// TIA Portal V17 export
// export: Created 2023-02-13T11:16:08.4914499Z, ExportSetting WithDefaults, DisplayName Totally Integrated Automation Portal, DisplayVersion V17, DisplayName TIA Portal Openness, DisplayVersion V17, DisplayName TIA Portal Teamcenter Gateway, DisplayVersion V17, DisplayName TIA Portal Version Control Interface, DisplayVersion V17, DisplayName SINAMICS Startdrive Advanced, DisplayVersion V17, DisplayName SINAMICS Startdrive G130, G150, S120, S150, SINAMICS MV, S210, DisplayVersion V17, DisplayName SINAMICS Startdrive G110M, G120, G120C, G120D, G120P, G115D, DisplayVersion V17, DisplayName STEP 7 Professional, DisplayVersion V17, DisplayName STEP 7 Safety, DisplayVersion V17, DisplayName WinCC Professional, DisplayVersion V17
FUNCTION_BLOCK "Alarm Flow Collector"   // FB211, LAD
{ S7_Optimized_Access := 'TRUE' }
VERSION : 0.1
// stored: AutoNumber false, IsIECCheckEnabled false, IsRetainMemResEnabled false, MemoryReserve 100, SetENOAutomatically false, UDAEnableTagReadback false
   VAR_INPUT
      Reset : Bool;
   END_VAR
   VAR
      alwaysON : Bool;
   END_VAR
   VAR RETAIN
      Param : Struct
         min_Flow : Struct
            ChiliAwetan1 : Real := 5.0;
            ChiliAwetan2 : Real := 5.0;
            ChiliAwetan3 : Real := 5.0;
            Tomato : Real := 5.0;
            ChiliFresh1 : Real := 5.0;
            ChiliFresh2 : Real := 5.0;
            ChiliFresh3 : Real := 5.0;
            Garlic : Real := 5.0;
            HW : Real := 5.0;
            Vinegar : Real := 5.0;
            Sugar : Real := 5.0;
            Salt : Real := 5.0;
            ProWater : Real := 5.0;
            Homomixer : Real := 5.0;
         END_STRUCT;
         timerMon : Struct
            ChiliAwetan1 : TON_TIME;
            ChiliAwetan2 : TON_TIME;
            ChiliAwetan3 : TON_TIME;
            Tomato : TON_TIME;
            ChiliFresh1 : TON_TIME;
            ChiliFresh2 : TON_TIME;
            ChiliFresh3 : TON_TIME;
            Garlic : TON_TIME;
            HW : TON_TIME;
            Vinegar : TON_TIME;
            Sugar : TON_TIME;
            Salt : TON_TIME;
            ProWater : TON_TIME;
            Homomixer : TON_TIME;
         END_STRUCT;
      END_STRUCT;
   END_VAR
   VAR
      AlarmFlow_Blend : Word;
   END_VAR
   // Param.timerMon.ChiliAwetan1.PT := T#20s;
   // Param.timerMon.ChiliAwetan2.PT := T#20s;
   // Param.timerMon.ChiliAwetan3.PT := T#20s;
   // Param.timerMon.Tomato.PT := T#20s;
   // Param.timerMon.ChiliFresh1.PT := T#20s;
   // Param.timerMon.ChiliFresh2.PT := T#20s;
   // Param.timerMon.ChiliFresh3.PT := T#20s;
   // Param.timerMon.Garlic.PT := T#20s;
   // Param.timerMon.HW.PT := T#20s;
   // Param.timerMon.Vinegar.PT := T#20s;
   // Param.timerMon.Sugar.PT := T#20s;
   // Param.timerMon.Salt.PT := T#20s;
   // Param.timerMon.ProWater.PT := T#20s;
   // Param.timerMon.Homomixer.PT := T#20s;
BEGIN

REGION Network 1: always ON
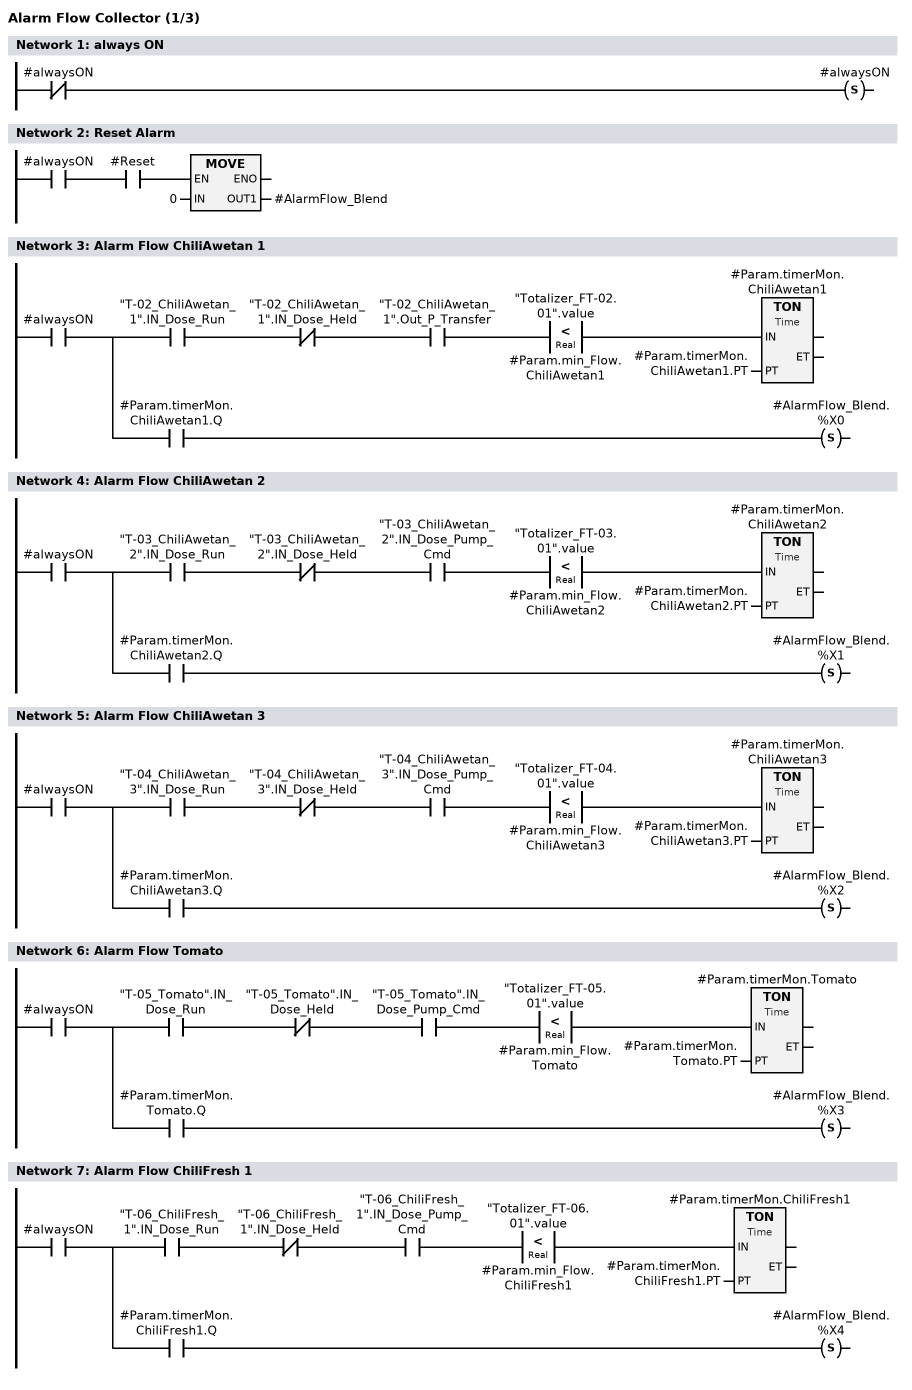
   RUNG wire#powerrail
      I_Contact( #alwaysON )
      S_Coil( #alwaysON )
   END_RUNG
   // the same network as SCL:
   IF NOT #alwaysON THEN #alwaysON := TRUE; END_IF;
END_REGION

REGION Network 2: Reset Alarm
   RUNG wire#powerrail
      Contact( #alwaysON )
      Contact( #Reset )
      Move(in := 0, out1 => #AlarmFlow_Blend)
   END_RUNG
   // the same network as SCL:
   IF #alwaysON AND #Reset THEN #AlarmFlow_Blend := 0; END_IF;
END_REGION

REGION Network 3: Alarm Flow ChiliAwetan 1
   RUNG wire#powerrail
      Contact( #alwaysON )
      wire#w1
      Contact( "T-02_ChiliAwetan_1".IN_Dose_Run )
      I_Contact( "T-02_ChiliAwetan_1".IN_Dose_Held )
      Contact( "T-02_ChiliAwetan_1".Out_P_Transfer )
      { S7_Templates := "SrcType := Real" } LT_Contact(in1 := "Totalizer_FT-02.01".value, in2 := #Param.min_Flow.ChiliAwetan1)
      { S7_Templates := "time_type := Time" } #Param.timerMon.ChiliAwetan1.TON(pt := #Param.timerMon.ChiliAwetan1.PT, et =>)
   END_RUNG
   RUNG wire#w1
      Contact( #Param.timerMon.ChiliAwetan1.Q )
      S_Coil( #AlarmFlow_Blend.%X0 )
   END_RUNG
   // the same network as SCL:
   #Param.timerMon.ChiliAwetan1.TON(IN := #alwaysON AND "T-02_ChiliAwetan_1".IN_Dose_Run AND NOT "T-02_ChiliAwetan_1".IN_Dose_Held AND "T-02_ChiliAwetan_1".Out_P_Transfer AND ("Totalizer_FT-02.01".value < #Param.min_Flow.ChiliAwetan1),
                           PT := #Param.timerMon.ChiliAwetan1.PT);
   IF #alwaysON AND #Param.timerMon.ChiliAwetan1.Q THEN #AlarmFlow_Blend.%X0 := TRUE; END_IF;
END_REGION

REGION Network 4: Alarm Flow ChiliAwetan 2
   RUNG wire#powerrail
      Contact( #alwaysON )
      wire#w1
      Contact( "T-03_ChiliAwetan_2".IN_Dose_Run )
      I_Contact( "T-03_ChiliAwetan_2".IN_Dose_Held )
      Contact( "T-03_ChiliAwetan_2".IN_Dose_Pump_Cmd )
      { S7_Templates := "SrcType := Real" } LT_Contact(in1 := "Totalizer_FT-03.01".value, in2 := #Param.min_Flow.ChiliAwetan2)
      { S7_Templates := "time_type := Time" } #Param.timerMon.ChiliAwetan2.TON(pt := #Param.timerMon.ChiliAwetan2.PT, et =>)
   END_RUNG
   RUNG wire#w1
      Contact( #Param.timerMon.ChiliAwetan2.Q )
      S_Coil( #AlarmFlow_Blend.%X1 )
   END_RUNG
   // the same network as SCL:
   #Param.timerMon.ChiliAwetan2.TON(IN := #alwaysON AND "T-03_ChiliAwetan_2".IN_Dose_Run AND NOT "T-03_ChiliAwetan_2".IN_Dose_Held AND "T-03_ChiliAwetan_2".IN_Dose_Pump_Cmd AND ("Totalizer_FT-03.01".value < #Param.min_Flow.ChiliAwetan2),
                           PT := #Param.timerMon.ChiliAwetan2.PT);
   IF #alwaysON AND #Param.timerMon.ChiliAwetan2.Q THEN #AlarmFlow_Blend.%X1 := TRUE; END_IF;
END_REGION

REGION Network 5: Alarm Flow ChiliAwetan 3
   RUNG wire#powerrail
      Contact( #alwaysON )
      wire#w1
      Contact( "T-04_ChiliAwetan_3".IN_Dose_Run )
      I_Contact( "T-04_ChiliAwetan_3".IN_Dose_Held )
      Contact( "T-04_ChiliAwetan_3".IN_Dose_Pump_Cmd )
      { S7_Templates := "SrcType := Real" } LT_Contact(in1 := "Totalizer_FT-04.01".value, in2 := #Param.min_Flow.ChiliAwetan3)
      { S7_Templates := "time_type := Time" } #Param.timerMon.ChiliAwetan3.TON(pt := #Param.timerMon.ChiliAwetan3.PT, et =>)
   END_RUNG
   RUNG wire#w1
      Contact( #Param.timerMon.ChiliAwetan3.Q )
      S_Coil( #AlarmFlow_Blend.%X2 )
   END_RUNG
   // the same network as SCL:
   #Param.timerMon.ChiliAwetan3.TON(IN := #alwaysON AND "T-04_ChiliAwetan_3".IN_Dose_Run AND NOT "T-04_ChiliAwetan_3".IN_Dose_Held AND "T-04_ChiliAwetan_3".IN_Dose_Pump_Cmd AND ("Totalizer_FT-04.01".value < #Param.min_Flow.ChiliAwetan3),
                           PT := #Param.timerMon.ChiliAwetan3.PT);
   IF #alwaysON AND #Param.timerMon.ChiliAwetan3.Q THEN #AlarmFlow_Blend.%X2 := TRUE; END_IF;
END_REGION

REGION Network 6: Alarm Flow Tomato
   RUNG wire#powerrail
      Contact( #alwaysON )
      wire#w1
      Contact( "T-05_Tomato".IN_Dose_Run )
      I_Contact( "T-05_Tomato".IN_Dose_Held )
      Contact( "T-05_Tomato".IN_Dose_Pump_Cmd )
      { S7_Templates := "SrcType := Real" } LT_Contact(in1 := "Totalizer_FT-05.01".value, in2 := #Param.min_Flow.Tomato)
      { S7_Templates := "time_type := Time" } #Param.timerMon.Tomato.TON(pt := #Param.timerMon.Tomato.PT, et =>)
   END_RUNG
   RUNG wire#w1
      Contact( #Param.timerMon.Tomato.Q )
      S_Coil( #AlarmFlow_Blend.%X3 )
   END_RUNG
   // the same network as SCL:
   #Param.timerMon.Tomato.TON(IN := #alwaysON AND "T-05_Tomato".IN_Dose_Run AND NOT "T-05_Tomato".IN_Dose_Held AND "T-05_Tomato".IN_Dose_Pump_Cmd AND ("Totalizer_FT-05.01".value < #Param.min_Flow.Tomato),
                           PT := #Param.timerMon.Tomato.PT);
   IF #alwaysON AND #Param.timerMon.Tomato.Q THEN #AlarmFlow_Blend.%X3 := TRUE; END_IF;
END_REGION

REGION Network 7: Alarm Flow ChiliFresh 1
   RUNG wire#powerrail
      Contact( #alwaysON )
      wire#w1
      Contact( "T-06_ChiliFresh_1".IN_Dose_Run )
      I_Contact( "T-06_ChiliFresh_1".IN_Dose_Held )
      Contact( "T-06_ChiliFresh_1".IN_Dose_Pump_Cmd )
      { S7_Templates := "SrcType := Real" } LT_Contact(in1 := "Totalizer_FT-06.01".value, in2 := #Param.min_Flow.ChiliFresh1)
      { S7_Templates := "time_type := Time" } #Param.timerMon.ChiliFresh1.TON(pt := #Param.timerMon.ChiliFresh1.PT, et =>)
   END_RUNG
   RUNG wire#w1
      Contact( #Param.timerMon.ChiliFresh1.Q )
      S_Coil( #AlarmFlow_Blend.%X4 )
   END_RUNG
   // the same network as SCL:
   #Param.timerMon.ChiliFresh1.TON(IN := #alwaysON AND "T-06_ChiliFresh_1".IN_Dose_Run AND NOT "T-06_ChiliFresh_1".IN_Dose_Held AND "T-06_ChiliFresh_1".IN_Dose_Pump_Cmd AND ("Totalizer_FT-06.01".value < #Param.min_Flow.ChiliFresh1),
                           PT := #Param.timerMon.ChiliFresh1.PT);
   IF #alwaysON AND #Param.timerMon.ChiliFresh1.Q THEN #AlarmFlow_Blend.%X4 := TRUE; END_IF;
END_REGION

REGION Network 8: Alarm Flow ChiliFresh 2
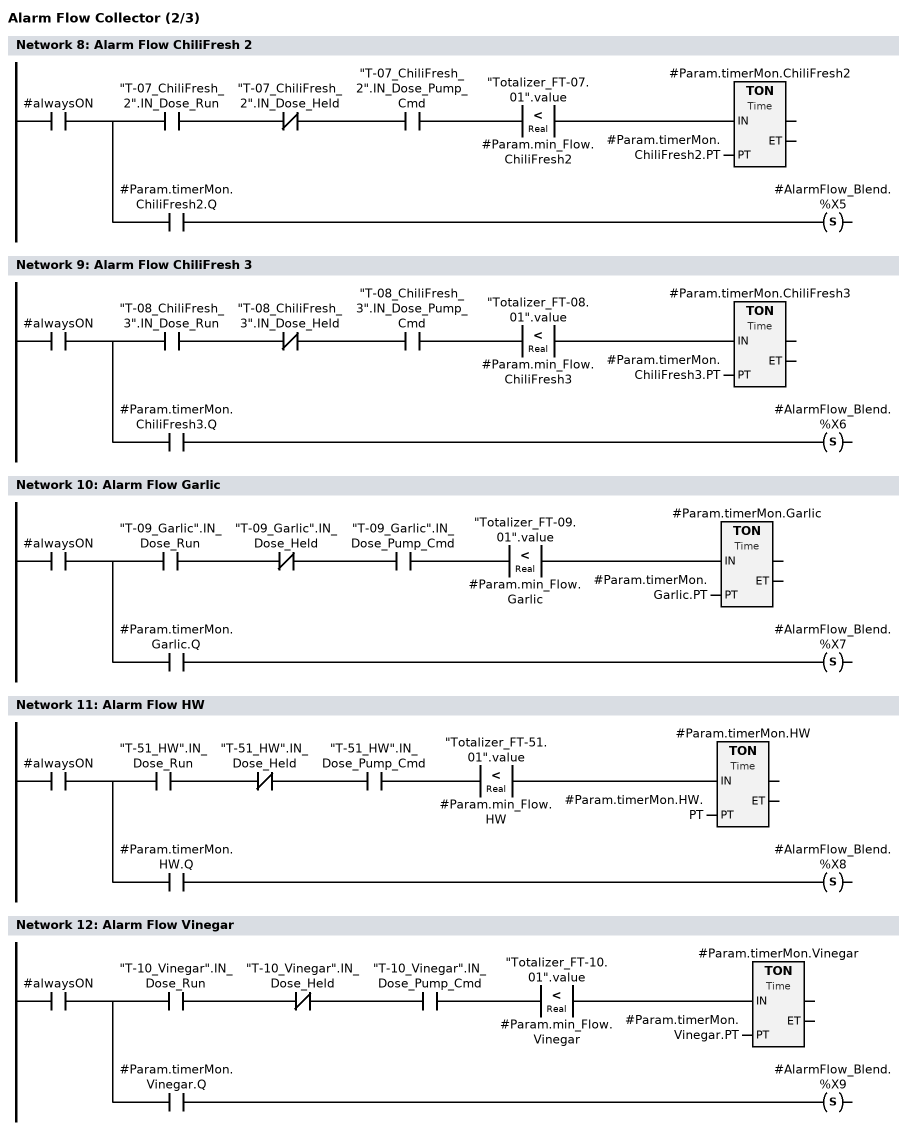
   RUNG wire#powerrail
      Contact( #alwaysON )
      wire#w1
      Contact( "T-07_ChiliFresh_2".IN_Dose_Run )
      I_Contact( "T-07_ChiliFresh_2".IN_Dose_Held )
      Contact( "T-07_ChiliFresh_2".IN_Dose_Pump_Cmd )
      { S7_Templates := "SrcType := Real" } LT_Contact(in1 := "Totalizer_FT-07.01".value, in2 := #Param.min_Flow.ChiliFresh2)
      { S7_Templates := "time_type := Time" } #Param.timerMon.ChiliFresh2.TON(pt := #Param.timerMon.ChiliFresh2.PT, et =>)
   END_RUNG
   RUNG wire#w1
      Contact( #Param.timerMon.ChiliFresh2.Q )
      S_Coil( #AlarmFlow_Blend.%X5 )
   END_RUNG
   // the same network as SCL:
   #Param.timerMon.ChiliFresh2.TON(IN := #alwaysON AND "T-07_ChiliFresh_2".IN_Dose_Run AND NOT "T-07_ChiliFresh_2".IN_Dose_Held AND "T-07_ChiliFresh_2".IN_Dose_Pump_Cmd AND ("Totalizer_FT-07.01".value < #Param.min_Flow.ChiliFresh2),
                           PT := #Param.timerMon.ChiliFresh2.PT);
   IF #alwaysON AND #Param.timerMon.ChiliFresh2.Q THEN #AlarmFlow_Blend.%X5 := TRUE; END_IF;
END_REGION

REGION Network 9: Alarm Flow ChiliFresh 3
   RUNG wire#powerrail
      Contact( #alwaysON )
      wire#w1
      Contact( "T-08_ChiliFresh_3".IN_Dose_Run )
      I_Contact( "T-08_ChiliFresh_3".IN_Dose_Held )
      Contact( "T-08_ChiliFresh_3".IN_Dose_Pump_Cmd )
      { S7_Templates := "SrcType := Real" } LT_Contact(in1 := "Totalizer_FT-08.01".value, in2 := #Param.min_Flow.ChiliFresh3)
      { S7_Templates := "time_type := Time" } #Param.timerMon.ChiliFresh3.TON(pt := #Param.timerMon.ChiliFresh3.PT, et =>)
   END_RUNG
   RUNG wire#w1
      Contact( #Param.timerMon.ChiliFresh3.Q )
      S_Coil( #AlarmFlow_Blend.%X6 )
   END_RUNG
   // the same network as SCL:
   #Param.timerMon.ChiliFresh3.TON(IN := #alwaysON AND "T-08_ChiliFresh_3".IN_Dose_Run AND NOT "T-08_ChiliFresh_3".IN_Dose_Held AND "T-08_ChiliFresh_3".IN_Dose_Pump_Cmd AND ("Totalizer_FT-08.01".value < #Param.min_Flow.ChiliFresh3),
                           PT := #Param.timerMon.ChiliFresh3.PT);
   IF #alwaysON AND #Param.timerMon.ChiliFresh3.Q THEN #AlarmFlow_Blend.%X6 := TRUE; END_IF;
END_REGION

REGION Network 10: Alarm Flow Garlic
   RUNG wire#powerrail
      Contact( #alwaysON )
      wire#w1
      Contact( "T-09_Garlic".IN_Dose_Run )
      I_Contact( "T-09_Garlic".IN_Dose_Held )
      Contact( "T-09_Garlic".IN_Dose_Pump_Cmd )
      { S7_Templates := "SrcType := Real" } LT_Contact(in1 := "Totalizer_FT-09.01".value, in2 := #Param.min_Flow.Garlic)
      { S7_Templates := "time_type := Time" } #Param.timerMon.Garlic.TON(pt := #Param.timerMon.Garlic.PT, et =>)
   END_RUNG
   RUNG wire#w1
      Contact( #Param.timerMon.Garlic.Q )
      S_Coil( #AlarmFlow_Blend.%X7 )
   END_RUNG
   // the same network as SCL:
   #Param.timerMon.Garlic.TON(IN := #alwaysON AND "T-09_Garlic".IN_Dose_Run AND NOT "T-09_Garlic".IN_Dose_Held AND "T-09_Garlic".IN_Dose_Pump_Cmd AND ("Totalizer_FT-09.01".value < #Param.min_Flow.Garlic),
                           PT := #Param.timerMon.Garlic.PT);
   IF #alwaysON AND #Param.timerMon.Garlic.Q THEN #AlarmFlow_Blend.%X7 := TRUE; END_IF;
END_REGION

REGION Network 11: Alarm Flow HW
   RUNG wire#powerrail
      Contact( #alwaysON )
      wire#w1
      Contact( "T-51_HW".IN_Dose_Run )
      I_Contact( "T-51_HW".IN_Dose_Held )
      Contact( "T-51_HW".IN_Dose_Pump_Cmd )
      { S7_Templates := "SrcType := Real" } LT_Contact(in1 := "Totalizer_FT-51.01".value, in2 := #Param.min_Flow.HW)
      { S7_Templates := "time_type := Time" } #Param.timerMon.HW.TON(pt := #Param.timerMon.HW.PT, et =>)
   END_RUNG
   RUNG wire#w1
      Contact( #Param.timerMon.HW.Q )
      S_Coil( #AlarmFlow_Blend.%X8 )
   END_RUNG
   // the same network as SCL:
   #Param.timerMon.HW.TON(IN := #alwaysON AND "T-51_HW".IN_Dose_Run AND NOT "T-51_HW".IN_Dose_Held AND "T-51_HW".IN_Dose_Pump_Cmd AND ("Totalizer_FT-51.01".value < #Param.min_Flow.HW),
                          PT := #Param.timerMon.HW.PT);
   IF #alwaysON AND #Param.timerMon.HW.Q THEN #AlarmFlow_Blend.%X8 := TRUE; END_IF;
END_REGION

REGION Network 12: Alarm Flow Vinegar
   RUNG wire#powerrail
      Contact( #alwaysON )
      wire#w1
      Contact( "T-10_Vinegar".IN_Dose_Run )
      I_Contact( "T-10_Vinegar".IN_Dose_Held )
      Contact( "T-10_Vinegar".IN_Dose_Pump_Cmd )
      { S7_Templates := "SrcType := Real" } LT_Contact(in1 := "Totalizer_FT-10.01".value, in2 := #Param.min_Flow.Vinegar)
      { S7_Templates := "time_type := Time" } #Param.timerMon.Vinegar.TON(pt := #Param.timerMon.Vinegar.PT, et =>)
   END_RUNG
   RUNG wire#w1
      Contact( #Param.timerMon.Vinegar.Q )
      S_Coil( #AlarmFlow_Blend.%X9 )
   END_RUNG
   // the same network as SCL:
   #Param.timerMon.Vinegar.TON(IN := #alwaysON AND "T-10_Vinegar".IN_Dose_Run AND NOT "T-10_Vinegar".IN_Dose_Held AND "T-10_Vinegar".IN_Dose_Pump_Cmd AND ("Totalizer_FT-10.01".value < #Param.min_Flow.Vinegar),
                           PT := #Param.timerMon.Vinegar.PT);
   IF #alwaysON AND #Param.timerMon.Vinegar.Q THEN #AlarmFlow_Blend.%X9 := TRUE; END_IF;
END_REGION

REGION Network 13: Alarm Flow Sugar
END_REGION

REGION Network 14: Alarm Flow Salt
END_REGION

REGION Network 15: Alarm Flow Prowater
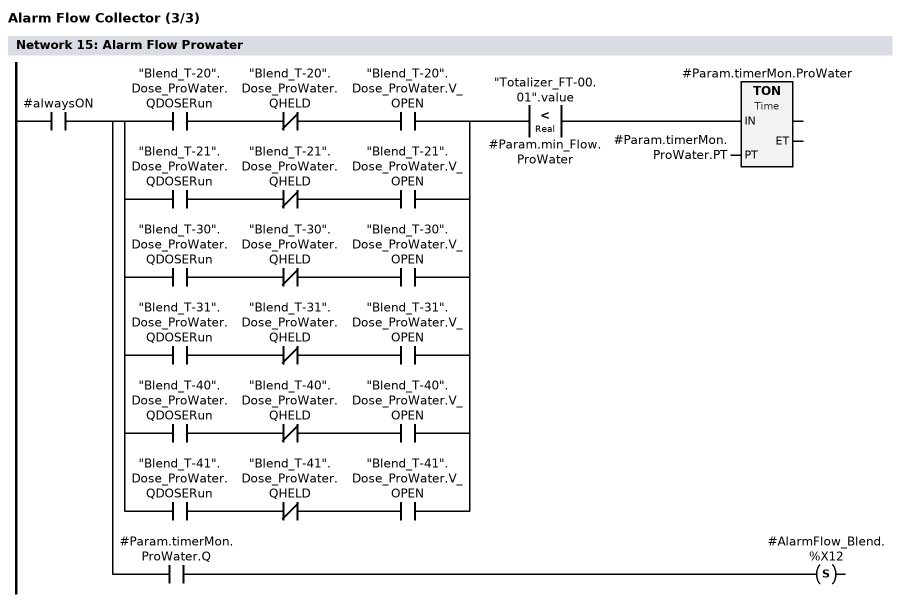
   RUNG wire#powerrail
      Contact( #alwaysON )
      wire#w1
      Contact( "Blend_T-20".Dose_ProWater.QDOSERun )
      I_Contact( "Blend_T-20".Dose_ProWater.QHELD )
      Contact( "Blend_T-20".Dose_ProWater.V_OPEN )
      wire#w2
      { S7_Templates := "SrcType := Real" } LT_Contact(in1 := "Totalizer_FT-00.01".value, in2 := #Param.min_Flow.ProWater)
      { S7_Templates := "time_type := Time" } #Param.timerMon.ProWater.TON(pt := #Param.timerMon.ProWater.PT, et =>)
   END_RUNG
   RUNG wire#w1
      Contact( "Blend_T-21".Dose_ProWater.QDOSERun )
      I_Contact( "Blend_T-21".Dose_ProWater.QHELD )
      Contact( "Blend_T-21".Dose_ProWater.V_OPEN )
   END_RUNG wire#w2
   RUNG wire#w1
      Contact( "Blend_T-30".Dose_ProWater.QDOSERun )
      I_Contact( "Blend_T-30".Dose_ProWater.QHELD )
      Contact( "Blend_T-30".Dose_ProWater.V_OPEN )
   END_RUNG wire#w2
   RUNG wire#w1
      Contact( "Blend_T-31".Dose_ProWater.QDOSERun )
      I_Contact( "Blend_T-31".Dose_ProWater.QHELD )
      Contact( "Blend_T-31".Dose_ProWater.V_OPEN )
   END_RUNG wire#w2
   RUNG wire#w1
      Contact( "Blend_T-40".Dose_ProWater.QDOSERun )
      I_Contact( "Blend_T-40".Dose_ProWater.QHELD )
      Contact( "Blend_T-40".Dose_ProWater.V_OPEN )
   END_RUNG wire#w2
   RUNG wire#w1
      Contact( "Blend_T-41".Dose_ProWater.QDOSERun )
      I_Contact( "Blend_T-41".Dose_ProWater.QHELD )
      Contact( "Blend_T-41".Dose_ProWater.V_OPEN )
   END_RUNG wire#w2
   RUNG wire#w1
      Contact( #Param.timerMon.ProWater.Q )
      S_Coil( #AlarmFlow_Blend.%X12 )
   END_RUNG
   // the same network as SCL:
   #Param.timerMon.ProWater.TON(IN := #alwaysON AND (("Blend_T-20".Dose_ProWater.QDOSERun AND NOT "Blend_T-20".Dose_ProWater.QHELD AND "Blend_T-20".Dose_ProWater.V_OPEN) OR ("Blend_T-21".Dose_ProWater.QDOSERun AND NOT "Blend_T-21".Dose_ProWater.QHELD AND "Blend_T-21".Dose_ProWater.V_OPEN) OR ("Blend_T-30".Dose_ProWater.QDOSERun AND NOT "Blend_T-30".Dose_ProWater.QHELD AND "Blend_T-30".Dose_ProWater.V_OPEN) OR ("Blend_T-31".Dose_ProWater.QDOSERun AND NOT "Blend_T-31".Dose_ProWater.QHELD AND "Blend_T-31".Dose_ProWater.V_OPEN) OR ("Blend_T-40".Dose_ProWater.QDOSERun AND NOT "Blend_T-40".Dose_ProWater.QHELD AND "Blend_T-40".Dose_ProWater.V_OPEN) OR ("Blend_T-41".Dose_ProWater.QDOSERun AND NOT "Blend_T-41".Dose_ProWater.QHELD AND "Blend_T-41".Dose_ProWater.V_OPEN)) AND ("Totalizer_FT-00.01".value < #Param.min_Flow.ProWater),
                           PT := #Param.timerMon.ProWater.PT);
   IF #alwaysON AND #Param.timerMon.ProWater.Q THEN #AlarmFlow_Blend.%X12 := TRUE; END_IF;
END_REGION
END_FUNCTION_BLOCK
